(* Enums for setting proper action in proper request. Used only internaly for FB_CR800Ethercat *) 
//{attribute 'qualified_only'}
//{attribute 'strict'}
TYPE E_RobotSystemActions :
(
	SET_INITIAL_PARAMETERS 	:= 0, 
	DO_HOMING 				:= 1,
	GO_AUTO					:= 11,
	UPDATE_RECIPIES 		:= 12	
)UINT;
END_TYPE

(* stored: Version 1.1.0.1, ProductVersion 3.1.4024.9
   DUT E_RobotSystemActions: Id {07de02da-a20d-419c-86bf-419c29639074} *)
